(* CODESYS project Alarming.library
   Company: Ziga Javornik
   DefaultNamespace: ZigaLibs.Alarming
   Version: 0.0.3.1
   Placeholder: ZigaLibs.Alarming
   Author: Ziga Javornik
   Description: A library for alarm management. Uses ZigaLibs_Logging to create the alarm logs files.
   Title: ZigaLibs.Alarming

Project tree, tasks and I/O mapping:
  libraries: Tc2_Standard, 3.4.5.0 (Beckhoff Automation GmbH); Tc2_System, 3.6.4.0 (Beckhoff Automation GmbH); Tc2_Utilities, * (Beckhoff Automation GmbH); Tc3_Module, 3.4.5.0 (Beckhoff Automation GmbH); TcUnit, 1.3.1 (www.tcunit.org); ZigaLibs.Core, 0.0.3.7 (Ziga Javornik); ZigaLibs.Logging, 0.0.4.1 (Ziga Javornik)
  GVLs/
  SOURCE/
    AlarmManager/
      Actions - fluent/
        function block FB_AlarmActionBuilder [ST]: Acknowledge, ById, ByName, Deactivate, DoAction, FB_init, Raise, SelectedAlarm
        interface I_AlarmActionBy: ById, ByName
        interface I_AlarmActions: Acknowledge, Deactivate, Raise
      DUTs/
        function block AlarmsArray [ST]: FB_exit, AddNew, Clear, Create, GetPtr, Remove, Set, NumberOfAlarms
        data type ST_AlarmInfo
        data type ST_AlarmTimeInfos
      data type E_AlarmLevel
      function block FB_AlarmManager [ST]: FB_init, AcknowledgeAlarmById, DeactivateAlarmById, RaiseAlarmById, AcknowledgeAlarmByName, DeactivateAlarmByName, RaiseAlarmByName, AcknowledgeAlarm, DeactivateAlarm, DeactivateAllAlarms, GetAlarmIndex, RaiseAlarm, AcknowledgeAllAlarms, Actions, DeleteAlarm, DeleteAll, GetAlarmById, GetAlarmByName, RegisterAlarm, ActiveAlarmsCount, Enable, RegisteredAlarmsCount, UnacknowledgedAlarmsCount
      interface I_AlarmManager: AcknowledgeAllAlarms, Actions, ActiveAlarmsCount, DeleteAlarm, DeleteAll, Enable, GetAlarmById, GetAlarmByName, RegisterAlarm, RegisteredAlarmsCount, UnacknowledgedAlarmsCount
  TESTS/
    Test suites/
      function block FB_AlarmManager_Tests [ST]: Test00_RegisterAlarms, Test01_ActivateNewAlarm_ExpectUnacknowledgedActiveAlarm, Test02_AcknowledgeActiveAlarm_ExpectActiveAcknowledged, Test03_ActivateExistingAlarm_ExpectSameActiveAlarmCount, Test04_DeactivateAlarm_ExpectNotActiveAcknowledged, Test05_AcknowlidgeInactiveAlarm_ExpectAcknowledgedNotActive, Test06_DisableManager_ExpectNoActiveAlarms, Test07_AcknowledgeAllAlarms_ExpectActiveAlarmsUnchanged, Test08_ActivateByName, Test09_DeactivateByName, Test10_AcknowledgeByName, Test11_GetAlarmByName, Test12_GetAlarmById, Test13_ActivateById, Test14_DeactivateById, Test15_AcknowledgeById, Test16_TimeInfos, Test17_RaiseUnexisitngAlarm_ExpectNoNewAlarmsActive, Test18_DeleteAlarm_ExpectPreviousAlarmsStillExist, Test19_DeleteUnexistingAlarm_ExpectNoChangesToExistingAlarms, Test20_DeleteAll
    program PRG_TESTS [ST]
*)

// SOURCE/AlarmManager/DUTs/ST_AlarmInfo
// Alarm information structure, containing all the informations requoired
TYPE ST_AlarmInfo :
STRUCT
	Name			: Tc2_System.T_MaxString;	// Name of the alarm
	Id				: T_ArrayIndexer;			// Id of the alarm
	Message			: Tc2_System.T_MaxString;	// Message of the alarm
	IsActive		: BOOL;						// Active state (TRUE = currently active, FALSE = not active)
	IsAcknowledged	: BOOL;						// Acknowledge state of the alarm
	Level			: E_AlarmLevel;				// Alarm level
	TimeInfos		: ST_AlarmTimeInfos;		// Time informations (activated, acknowldiged, deactivated)
END_STRUCT
END_TYPE

// SOURCE/AlarmManager/DUTs/ST_AlarmTimeInfos
// Provides time information for an alarm
TYPE ST_AlarmTimeInfos :
STRUCT
	Activated		: Tc2_Utilities.TIMESTRUCT;	// Time of alarm activation
	Deactivated		: Tc2_Utilities.TIMESTRUCT;	// Time of alarm deactiovation
	Acknowledged	: Tc2_Utilities.TIMESTRUCT;	// Time of alarm acknowlidgemenet
END_STRUCT
END_TYPE

// SOURCE/AlarmManager/E_AlarmLevel
{attribute 'qualified_only'}
{attribute 'strict'}
// Alarm level enumeration
TYPE E_AlarmLevel :
(
	NONE,
	INFO,
	WARNING,
	ERROR
);
END_TYPE

// SOURCE/AlarmManager/Actions - fluent/FB_AlarmActionBuilder
FUNCTION_BLOCK INTERNAL FB_AlarmActionBuilder IMPLEMENTS I_AlarmActionBy, I_AlarmActions
VAR
	_alarmAction 	: (ACTION_ACKNOWLEDGE, ACTTION_RAISE, ACTION_DEACTIVATE);
	_selectedAlarm	: REFERENCE TO ST_AlarmInfo;
	_alarmManager	: REFERENCE TO FB_AlarmManager;
END_VAR

METHOD Acknowledge : I_AlarmActionBy
VAR_INPUT
END_VAR
_alarmAction := ACTION_ACKNOWLEDGE;
Acknowledge := THIS^;
END_METHOD

// Executes the action by looking for the alarm with the provided ID
METHOD ById
VAR_INPUT
	Id	: T_ArrayIndexer;
END_VAR
VAR
	i	: T_ArrayIndexer;
END_VAR
IF NOT __ISVALIDREF(_alarmManager.GetAlarmById(Id)) THEN
	RETURN;
END_IF

_selectedAlarm REF= _alarmManager.GetAlarmById(Id);
DoAction();
END_METHOD

// Executes the action by looking for the alarm with the provided name
METHOD ByName
VAR_INPUT
	name	: Tc2_System.T_MaxString;
END_VAR

VAR_INST
	i	: T_ArrayIndexer;
END_VAR
IF NOT __ISVALIDREF(_alarmManager.GetAlarmByName(name)) THEN
	RETURN;
END_IF
_selectedAlarm REF= _alarmManager.GetAlarmByName(name);
DoAction();
END_METHOD

METHOD Deactivate : I_AlarmActionBy
VAR_INPUT
END_VAR
_alarmAction := ACTION_DEACTIVATE;
Deactivate := THIS^;
END_METHOD

METHOD PRIVATE DoAction
CASE _alarmAction OF
	ACTION_ACKNOWLEDGE:
		_alarmManager.AcknowledgeAlarm(_selectedAlarm);
	ACTTION_RAISE:
		_alarmManager.RaiseAlarm(_selectedAlarm);
	ACTION_DEACTIVATE:
		_alarmManager.DeactivateAlarm(_selectedAlarm);
END_CASE
END_METHOD

METHOD FB_init : BOOL
VAR_INPUT
	bInitRetains : BOOL; // if TRUE, the retain variables are initialized (warm start / cold start)
	bInCopyCode : BOOL;  // if TRUE, the instance afterwards gets moved into the copy code (online change)
	alarmManager	: REFERENCE TO FB_AlarmManager;
END_VAR
_alarmManager REF= alarmManager;
END_METHOD

METHOD Raise : I_AlarmActionBy
VAR_INPUT
END_VAR
_alarmAction := ACTTION_RAISE;
Raise := THIS^;
END_METHOD

PROPERTY SelectedAlarm : REFERENCE TO ST_AlarmInfo
GET
END_GET
END_PROPERTY

END_FUNCTION_BLOCK

// SOURCE/AlarmManager/Actions - fluent/I_AlarmActionBy
INTERFACE I_AlarmActionBy

// Executes the action by looking for the alarm with the provided ID
METHOD ById
VAR_INPUT
	Id	: T_ArrayIndexer;
END_VAR
END_METHOD

// Executes the action by looking for the alarm with the provided name
METHOD ByName
VAR_INPUT
	name	: Tc2_System.T_MaxString;
END_VAR
END_METHOD

END_INTERFACE

// SOURCE/AlarmManager/Actions - fluent/I_AlarmActions
INTERFACE I_AlarmActions

METHOD Acknowledge : I_AlarmActionBy
VAR_INPUT
END_VAR
END_METHOD

METHOD Deactivate : I_AlarmActionBy
VAR_INPUT
END_VAR
END_METHOD

METHOD Raise : I_AlarmActionBy
VAR_INPUT
END_VAR
END_METHOD

END_INTERFACE

// SOURCE/AlarmManager/FB_AlarmManager
(* 
Alarm manager function block. 
The body does not contain any logic, this it does not require being called.

====================================================
Constructor template:

(enable : , // Enables alarm generation
logger : , // If you do not want logging, simply set this variable to 0, internal checks will ommit any logging.
timeProvider : ); // Date time provider.*)

{attribute 'no_explicit_call' := 'Body contains no logic, calling methods only allowed.'}
FUNCTION_BLOCK FB_AlarmManager IMPLEMENTS I_AlarmManager

VAR
	_enable						: BOOL;
	_stringBuilder				: ZigaLibs_Core.FB_StringBuilder;
	_dateTime					: ZigaLibs_Core.I_LocalSystemTimeProvider;
	_activeAlarmCount			: UINT;
	_logger						: REFERENCE TO ZigaLibs_Logging.I_Logger; // If provided, logging will be used.
	_emptyAlarm					: ST_AlarmInfo;
	_registeredAlarmsCount		: UDINT;
	_alarmActionBuilder			: FB_AlarmActionBuilder(THIS^);
	_alarms						: AlarmsArray;
END_VAR

METHOD FB_init : BOOL
VAR_INPUT
	bInitRetains 	: BOOL; // if TRUE, the retain variables are initialized (warm start / cold start)
	bInCopyCode 	: BOOL;  // if TRUE, the instance afterwards gets moved into the copy code (online change)
	enable			: BOOL;	// Enables alarm generation
	logger			: REFERENCE TO ZigaLibs_Logging.I_Logger; // If you do not want logging, simply set this variable to 0, internal checks will ommit any logging.
	timeProvider	: ZigaLibs_Core.I_LocalSystemTimeProvider;	// Date time provider.
END_VAR
_enable := enable;
_logger REF= logger;
_dateTime := timeProvider;
END_METHOD

(* Acknowledges the alarm with the provided id*)
METHOD INTERNAL AcknowledgeAlarmById
VAR_INPUT
	nId	: T_ArrayIndexer;
END_VAR

VAR
	foundAlarm	: ST_AlarmInfo;
END_VAR
IF NOT __ISVALIDREF(GetAlarmById(nID := nId)) THEN
	RETURN;
END_IF

foundAlarm := GetAlarmById(nID := nId);
IF foundAlarm.Id = nId THEN
	AcknowledgeAlarm(alarm := GetAlarmById(nID := nId));
	RETURN;
END_IF
END_METHOD

(* Deactivates the alarm with the provided Id (if it exists).*)
METHOD INTERNAL DeactivateAlarmById
VAR_INPUT
	(* Alarm id to be deactivated.*)
	nId	: T_ArrayIndexer;
END_VAR

VAR
	foundAlarm	 : ST_AlarmInfo;
END_VAR
IF NOT __ISVALIDREF(GetAlarmById(nID := nId)) THEN
	RETURN;
END_IF

foundAlarm := GetAlarmById(nID := nId);

IF foundAlarm.Id = nId THEN
	DeactivateAlarm(alarm := GetAlarmById(nID := nId));
	RETURN;
END_IF
END_METHOD

(* Activates the alarm with the provided Id (if it exists)*)
METHOD INTERNAL RaiseAlarmById
VAR_INPUT
	(* Alarm id to be activated*)
	nId	: T_ArrayIndexer;
END_VAR

VAR
	foundAlarm	 : ST_AlarmInfo;
END_VAR
IF NOT __ISVALIDREF(GetAlarmById(nID := nId)) THEN
	RETURN;
END_IF

foundAlarm := GetAlarmById(nID := nId);
IF foundAlarm.Id = nId THEN
	RaiseAlarm(alarm := GetAlarmById(nID := nId));
	RETURN;
END_IF
END_METHOD

(* Acknowledges the alarm with the provided name.*)
METHOD INTERNAL AcknowledgeAlarmByName
VAR_INPUT
	sName	: Tc2_System.T_MaxString;
END_VAR

VAR
	foundAlarm	: ST_AlarmInfo;
END_VAR
IF NOT __ISVALIDREF(GetAlarmByName(sName := sName)) THEN
	RETURN;
END_IF

foundAlarm := GetAlarmByName(sName := sName);
IF foundAlarm.Name = sName THEN
	AcknowledgeAlarm(alarm := GetAlarmByName(sName := sName));
	RETURN;
END_IF
END_METHOD

(* Deactivates the alarm with the provided name (if it exists)*)
METHOD INTERNAL DeactivateAlarmByName
VAR_INPUT
	(* Alarm name to be deactivated.*)
	sName	: Tc2_System.T_MaxString;
END_VAR

VAR
	foundAlarm	 : ST_AlarmInfo;
END_VAR
IF NOT __ISVALIDREF(GetAlarmByName(sName := sName)) THEN
	RETURN;
END_IF

foundAlarm := GetAlarmByName(sName := sName);
IF foundAlarm.Name = sName THEN
	DeactivateAlarm(alarm := GetAlarmByName(sName := sName));
	RETURN;
END_IF
END_METHOD

(* Activates the alarm with the provided name*)
METHOD INTERNAL RaiseAlarmByName
VAR_INPUT
	(* Alarm name to be actived*)
	sName	: Tc2_System.T_MaxString;
END_VAR

VAR
	foundAlarm	 : ST_AlarmInfo;
END_VAR
IF NOT __ISVALIDREF(GetAlarmByName(sName := sName)) THEN
	RETURN;
END_IF

foundAlarm := GetAlarmByName(sName := sName);
IF foundAlarm.Name = sName THEN
	RaiseAlarm(alarm := GetAlarmByName(sName := sName));
	RETURN;
END_IF
END_METHOD

METHOD INTERNAL AcknowledgeAlarm
VAR_INPUT
	alarm : REFERENCE TO ST_AlarmInfo;
END_VAR
IF alarm.IsAcknowledged THEN
	RETURN;
END_IF

alarm.IsAcknowledged := TRUE;
alarm.TimeInfos.Acknowledged := _dateTime.CurrentTime.Value;

IF __ISVALIDREF(_logger) THEN 
	_logger.LogInfo(_stringBuilder.Reset()
		.AddString('Alarm ')
		.AddWithDblQuotationMarks(str := alarm.Name)
		.AddString(' with Id ')
		.AddWithDblQuotationMarks(str := TO_STRING(alarm.Id))
		.AddString(' acknowledged.')
		.Create());
END_IF
END_METHOD

METHOD INTERNAL DeactivateAlarm
VAR_INPUT
	alarm : REFERENCE TO ST_AlarmInfo;
END_VAR
IF NOT alarm.IsActive THEN
	RETURN;
END_IF

alarm.IsActive := FALSE;
alarm.TimeInfos.Deactivated := _dateTime.CurrentTime.Value;
_activeAlarmCount := _activeAlarmCount - 1;

IF __ISVALIDREF(_logger) THEN
	_logger.LogInfo(_stringBuilder
		.Reset()
		.AddString('Alarm ')
		.AddWithDblQuotationMarks(str := alarm.Name)
		.AddString(' with Id ')
		.AddWithDblQuotationMarks(str := TO_STRING(alarm.Id))
		.AddString(' deactivated.')
		.Create());
END_IF
END_METHOD

METHOD PRIVATE DeactivateAllAlarms

VAR
	alarmIndex	: T_ArrayIndexer;
END_VAR
FOR alarmIndex := 0 TO _alarms.NumberOfAlarms BY 1 DO
	IF _alarms.GetPtr(alarmIndex) <> 0 AND_THEN _alarms.GetPtr(alarmIndex)^.IsActive THEN
		DeactivateAlarm(_alarms.GetPtr(alarmIndex)^);
	END_IF
END_FOR
END_METHOD

METHOD PRIVATE GetAlarmIndex : DINT
VAR_INPUT
	id	: DINT;
END_VAR
VAR_OUTPUT
	exists	: BOOL;
END_VAR
VAR
	alarmIndex	: DINT;
	alarmPtr	: POINTER TO ST_AlarmInfo;
END_VAR
FOR alarmIndex := 0 TO _alarms.NumberOfAlarms - 1 BY 1 DO
	alarmPtr := _alarms.GetPtr(alarmIndex);
	IF alarmPtr <> 0 AND_THEN alarmPtr^.Id = id THEN 
		GetAlarmIndex := alarmIndex;
		exists := TRUE;
		RETURN;
	END_IF
END_FOR
END_METHOD

METHOD INTERNAL RaiseAlarm
VAR_INPUT
	alarm : REFERENCE TO ST_AlarmInfo;
END_VAR
VAR
	message	: Tc2_System.T_MaxString;
END_VAR
IF alarm.IsActive OR NOT _enable THEN
	RETURN;
END_IF

_activeAlarmCount := _activeAlarmCount + 1;
alarm.IsActive := TRUE;
alarm.IsAcknowledged := FALSE;
Tc2_System.MEMSET(
	destAddr := ADR(alarm.TimeInfos),
	fillByte := 0,
	n := SIZEOF(alarm.TimeInfos));
	
alarm.TimeInfos.Activated := _dateTime.CurrentTime.Value;

IF __ISVALIDREF(_logger) THEN
	message := _stringBuilder.Reset()
		.AddString('Alarm ')
		.AddWithDblQuotationMarks(str := alarm.Name)
		.AddString(' with Id ')
		.AddWithDblQuotationMarks(str := TO_STRING(alarm.Id))
		.AddString(' actived! ')
		.AddString(alarm.Message)
		.Create();
		
	CASE alarm.Level OF 
		E_AlarmLevel.NONE: _logger.LogDefault(message := message);
		E_AlarmLevel.INFO: _logger.LogInfo(message := message);
		E_AlarmLevel.WARNING: _logger.LogWarning(message := message);
		E_AlarmLevel.ERROR: _logger.LogError(message := message);
	END_CASE
END_IF
END_METHOD

(* Acknowledges all uacknowledged alarms.*)
METHOD AcknowledgeAllAlarms
VAR
	alarmIndex	: T_ArrayIndexer;
END_VAR
FOR alarmIndex := 0 TO _alarms.NumberOfAlarms - 1 BY 1 DO
	IF _alarms.GetPtr(alarmIndex) <> 0 THEN 
		AcknowledgeAlarm(_alarms.GetPtr(alarmIndex)^);
	END_IF
END_FOR
END_METHOD

// Provides access to action builder with fluent approach.
METHOD PUBLIC Actions : I_AlarmActions
VAR_INPUT
END_VAR
Actions := _alarmActionBuilder;
END_METHOD

(* Deletes the alarm with the provided id.*)
METHOD DeleteAlarm
VAR_INPUT
	id	: DINT;
END_VAR
VAR
	exists	: BOOL;
	index	: DINT;
	alarm	: POINTER TO ST_AlarmInfo;
END_VAR
index := THIS^.GetAlarmIndex(id, exists => exists);
IF exists THEN
	alarm := _alarms.GetPtr(index);
	IF alarm^.IsActive THEN
		_activeAlarmCount := _activeAlarmCount - 1;
	END_IF
	_alarms.Remove(index);
END_IF
END_METHOD

(* Deletes all existing alarms from the memory*)
METHOD DeleteAll
_alarms.Clear();
_activeAlarmCount := 0;
END_METHOD

(* Gets the alarm with the provided id. 
 If no mathching alarm exists, an invalid reference will be returned - check by using __ISVALIDREF() for any further operations!.*)
METHOD GetAlarmById : REFERENCE TO ST_AlarmInfo
VAR_INPUT
	(* Id of the alarm.*)
	nID	: T_ArrayIndexer;
END_VAR

VAR
	index		: ZigaLibs_Core.T_ArrayIndexer;
	alarmPtr	: POINTER TO ST_AlarmInfo;
END_VAR
FOR index := 0 TO _alarms.NumberOfAlarms - 1 BY 1 DO
	alarmPtr := _alarms.GetPtr(index);
	IF alarmPtr <> 0 AND_THEN alarmPtr^.Id = nId THEN
		GetAlarmById REF= _alarms.GetPtr(index)^;
		RETURN;
	END_IF
END_FOR
END_METHOD

(* Gets the alarm with the provided name. 
 If no mathching alarm exists, an empty alarm is returned.*)
METHOD GetAlarmByName : REFERENCE TO ST_AlarmInfo
VAR_INPUT
	(* Name of the alarm*)
	sName	: Tc2_System.T_MaxString;
END_VAR

VAR
	index	 : T_ArrayIndexer;
END_VAR
FOR index := 0 TO _alarms.NumberOfAlarms - 1 BY 1 DO
	IF _alarms.GetPtr(index) <> 0 AND_THEN _alarms.GetPtr(index)^.Name = sName THEN
		GetAlarmByName REF= _alarms.GetPtr(index)^;
		RETURN;
	END_IF
END_FOR
END_METHOD

(* Registers a new alarm with the provided information. 
 Returns TRUE if new alarm was registered or false if not (alarm buffer is full or the id already exists)*)
METHOD RegisterAlarm : BOOL
VAR_INPUT
	(* Alarm ID*)
	Id	: T_ArrayIndexer;
	(* Alarm name*)
	Name	: Tc2_System.T_MaxString;
	(* Message when the alarm occurrs*)
	Message	: Tc2_System.T_MaxString;
	(* Alarm level *)
	Level	: E_AlarmLevel;				
END_VAR

VAR
	alarmIndex	: T_ArrayIndexer;
	alarm		:  ST_AlarmInfo;
END_VAR
// IF an alar is found, check the id and return.
IF __ISVALIDREF(GetAlarmById(nID := Id)) AND_THEN GetAlarmById(nID := Id).Id = Id 
THEN
	RETURN;
END_IF

// Create the alarm
alarm.Id := Id;
alarm.Name := Name;
alarm.Message := Message;
alarm.IsAcknowledged := TRUE;
alarm.Level := Level;
_alarms.AddNew(alarm);
RegisterAlarm := TRUE;
END_METHOD

{attribute 'monitoring':='call'}
(* Gets the total count of currently active alarms*)
PROPERTY ActiveAlarmsCount : UINT
GET
ActiveAlarmsCount := _activeAlarmCount;
END_GET
END_PROPERTY

{attribute 'monitoring':='call'}
(* Gets or sets if alarm manager is enabled or not. When disabled, all active alarms will become inactive!*)
PROPERTY Enable : BOOL
GET
Enable := _enable;
END_GET
SET
IF NOT Enable AND _enable THEN 
	IF __ISVALIDREF(_logger) THEN
		_logger.LogInfo('Alarms are now disabled.');
	END_IF
	DeactivateAllAlarms();
	AcknowledgeAllAlarms();
ELSIF Enable AND NOT _enable THEN
	IF __ISVALIDREF(_logger) THEN
		_logger.LogInfo('Alarms are now enabled.');
	END_IF
END_IF

_enable := Enable;
END_SET
END_PROPERTY

{attribute 'monitoring':='call'}
(* Gets the total number of alarms registered*)
PROPERTY RegisteredAlarmsCount : UDINT
GET
RegisteredAlarmsCount := DINT_TO_UDINT(_alarms.NumberOfAlarms);
END_GET
END_PROPERTY

{attribute 'monitoring':='call'}
(* Gets the current count of alarms that have not yet been acknowledged*)
PROPERTY UnacknowledgedAlarmsCount : UINT
GET
VAR
	alarmIndex		: T_ArrayIndexer;
	maxAlarmIndex	: T_ArrayIndexer;
	count			: UINT;
END_VAR
FOR alarmIndex := 0 TO _alarms.NumberOfAlarms - 1 BY 1 DO
	IF _alarms.GetPtr(alarmIndex) <> 0 AND_THEN NOT _alarms.GetPtr(alarmIndex)^.IsAcknowledged THEN
		count := count + 1;
	END_IF
END_FOR

UnacknowledgedAlarmsCount := count;
END_GET
END_PROPERTY

END_FUNCTION_BLOCK

// SOURCE/AlarmManager/I_AlarmManager
INTERFACE I_AlarmManager

// Acknowledges all uacknowledged alarms.
METHOD AcknowledgeAllAlarms
END_METHOD

// Provides access to action builder with fluent approach.
METHOD PUBLIC Actions : I_AlarmActions
VAR_INPUT
END_VAR
END_METHOD

{attribute 'monitoring':='call'}
// Gets the total count of currently active alarms
PROPERTY ActiveAlarmsCount : UINT
GET
END_GET
END_PROPERTY

// Deletes the alarm with the provided id.
METHOD DeleteAlarm
VAR_INPUT
	id	: DINT;
END_VAR
END_METHOD

// Deletes all existing alarms from the memory
METHOD DeleteAll
END_METHOD

{attribute 'monitoring':='call'}
// Gets or sets if alarm manager is enabled or not. When disabled, all active alarms will become inactive!
PROPERTY Enable : BOOL
GET
END_GET
SET
END_SET
END_PROPERTY

(* Gets the alarm with the provided id. 
 If no mathching alarm exists, an invalid reference will be returned - check by using __ISVALIDREF() for any further operations!.*)
METHOD GetAlarmById : REFERENCE TO ST_AlarmInfo
VAR_INPUT
	nID		: T_ArrayIndexer;	// Id of the alarm.
END_VAR
END_METHOD

// Gets the alarm with the provided name. 
// IF no mathching alarm exists, an invalid REFERENCE will be returned - check BY using __ISVALIDREF() FOR ANY further operations!.*)
METHOD GetAlarmByName : REFERENCE TO ST_AlarmInfo
VAR_INPUT
	sName	: Tc2_System.T_MaxString;	// Name of the alarm
END_VAR
END_METHOD

// Registers a new alarm with the provided information. 
// Returns TRUE if new alarm was registered or false if not
// Possible reasons for fail:
// - alarm buffer is full
// - the id already exists)
METHOD RegisterAlarm : BOOL
VAR_INPUT
	Id		: T_ArrayIndexer;			// Alarm ID
	Name	: Tc2_System.T_MaxString;	// Alarm name
	Message	: Tc2_System.T_MaxString;	// Message when the alarm occurrs
	Level	: E_AlarmLevel;				// Alarm level
END_VAR
END_METHOD

{attribute 'monitoring':='call'}
// Gets the total number of alarms registered
PROPERTY RegisteredAlarmsCount : UDINT
GET
END_GET
END_PROPERTY

{attribute 'monitoring':='call'}
// Gets the current count of alarms that have not yet been acknowledged
PROPERTY UnacknowledgedAlarmsCount : UINT
GET
END_GET
END_PROPERTY

END_INTERFACE

// SOURCE/AlarmManager/DUTs/AlarmsArray
// A dynamic collection of alarms as ST_AlarmInfo
FUNCTION_BLOCK AlarmsArray
VAR_INPUT
END_VAR
VAR_OUTPUT
END_VAR
VAR
	_malloc	: ZigaLibs_Core.FB_Malloc(0,0);
END_VAR

METHOD FB_exit : BOOL
VAR_INPUT
	bInCopyCode : BOOL; // if TRUE, the exit method is called for exiting an instance that is copied afterwards (online change).
END_VAR
_malloc.Free();
END_METHOD

// Adds a new alarm defintition to the collection
METHOD AddNew
VAR_INPUT
	alarm	: ST_AlarmInfo;
END_VAR
IF NOT _malloc.IsAllocated THEN
	THIS^.Create(1);
	THIS^.GetPtr(0)^ := alarm;
ELSE
	_malloc.Expand(1);
	_malloc.Set(_malloc.Properties.NumberOfElements - 1, alarm);
END_IF
END_METHOD

// Clear the entire collection of alarms
METHOD Clear
VAR_INPUT
END_VAR
_malloc.Free();
END_METHOD

// Creates a number of alarms defined by the count value
METHOD Create : BOOL
VAR_INPUT
	count	: dint;
END_VAR
Create := _malloc.Allocate(SIZEOF(ST_AlarmInfo), count);
END_METHOD

// Gets the pointer to the desired ST_AlarmInfo info at index
METHOD GetPtr : POINTER TO ST_AlarmInfo
VAR_INPUT
	index	: DINT;
END_VAR
GetPtr := _malloc.GetPtr(index);
END_METHOD

// Romves an alarm at the provided index
METHOD Remove
VAR_INPUT
	index	: DINT;
END_VAR
_malloc.Remove(index);
END_METHOD

// Sets the alarm at the index to the value provided in the alarm
METHOD Set : BOOL
VAR_INPUT
	index	: DINT;
	alarm	: REFERENCE TO ST_AlarmInfo;
END_VAR
Set := _malloc.Set(index := index, value := alarm);
END_METHOD

{attribute 'monitoring':='call'}
// Gets the total number of alarms in the collection
PROPERTY NumberOfAlarms : DINT
GET
NumberOfAlarms := _malloc.Properties.NumberOfElements;
END_GET
END_PROPERTY

END_FUNCTION_BLOCK

// TESTS/Test suites/FB_AlarmManager_Tests
FUNCTION_BLOCK INTERNAL FB_AlarmManager_Tests EXTENDS FB_TestSuite
VAR
	_dateTime	: ZigaLibs_Core.FB_LocalSystemTimeProvider;
	_alarmManager : FB_AlarmManager(
		enable := TRUE, // [BOOL] - Enables alarm generation
		logger := 0, // [REFERENCE TO ZigaLibs_Core.I_LoggerEx] - optional, logger.
		timeProvider := _dateTime); //[ZigaLibs_Core.I_LocalSystemTimeProvider] - required, date time provider.
END_VAR

_dateTime();
Test00_RegisterAlarms();
Test01_ActivateNewAlarm_ExpectUnacknowledgedActiveAlarm();
Test02_AcknowledgeActiveAlarm_ExpectActiveAcknowledged();
Test03_ActivateExistingAlarm_ExpectSameActiveAlarmCount();
Test04_DeactivateAlarm_ExpectNotActiveAcknowledged();
Test05_AcknowlidgeInactiveAlarm_ExpectAcknowledgedNotActive();
Test06_DisableManager_ExpectNoActiveAlarms();
Test07_AcknowledgeAllAlarms_ExpectActiveAlarmsUnchanged();
Test08_ActivateByName();
Test09_DeactivateByName();
Test10_AcknowledgeByName();
Test11_GetAlarmByName();
Test12_GetAlarmById();
Test13_ActivateById();
Test14_DeactivateById();
Test15_AcknowledgeById();
Test16_TimeInfos();
Test17_RaiseUnexisitngAlarm_ExpectNoNewAlarmsActive();
Test18_DeleteAlarm_ExpectPreviousAlarmsStillExist();
Test19_DeleteUnexistingAlarm_ExpectNoChangesToExistingAlarms();
Test20_DeleteAll();

METHOD Test00_RegisterAlarms
VAR_INPUT
END_VAR

VAR
	addAlarmIndex	: T_ArrayIndexer;
	alarm			: ST_AlarmInfo;
END_VAR
IF TcUnit.TEST_ORDERED('Test00_RegisterAlarms') THEN
	AssertEquals_UDINT(
		Actual := _alarmManager.RegisteredAlarmsCount,
		Expected := 0,
		Message := 'Before registering any alarms, the Registered count should be 0.');
	
	FOR addAlarmIndex := 1 TO 100 BY 1 DO
		AssertTrue(
			Condition := _alarmManager.RegisterAlarm(
				Id := addAlarmIndex,
				Message := Tc2_Standard.CONCAT('Alarm message', TO_STRING(addAlarmIndex)),
				Name := Tc2_Standard.CONCAT('Alarm name', TO_STRING(addAlarmIndex)),
				Level := E_AlarmLevel.INFO),
			Message := 'Registering alarm failed.');
			
		AssertEquals_UDINT(
			Actual := _alarmManager.RegisteredAlarmsCount,
			Expected := DINT_TO_UDINT(addAlarmIndex),
			Message := 'Registered alarm count is incorrect.');
			
		alarm := _alarmManager.GetAlarmById(nID := addAlarmIndex);
		AssertTrue(
			Condition := alarm.IsAcknowledged,
			Message := 'Newly registered alarm should be acknowledged by default, when created.');
	END_FOR
	
	AssertFalse(
		Condition := _alarmManager.RegisterAlarm(
			Id := 22,
			Message := CONCAT('Alarm message', TO_STRING(addAlarmIndex - 1)),
			Name := CONCAT('Alarm name', TO_STRING(addAlarmIndex - 1)),
			Level := E_AlarmLevel.INFO),
		Message := 'Registering an alarm with an existing id should not be possible.');
	
		
	TcUnit.TEST_FINISHED();
END_IF
END_METHOD

METHOD Test01_ActivateNewAlarm_ExpectUnacknowledgedActiveAlarm
VAR_INPUT
END_VAR

VAR
	currentAlarm	: ST_AlarmInfo;
END_VAR
IF TcUnit.TEST_ORDERED('Test01_ActivateNewAlarm_ExpectUnacknowledgedActiveAlarm') THEN
	_alarmManager.RaiseAlarmById(10);
	currentAlarm := _alarmManager.GetAlarmById(10);
	
	AssertEquals_BOOL(
		Actual := currentAlarm.IsActive,
		Expected := TRUE,
		Message := 'Alarm activation failed.');
		
	AssertEquals_BOOL(
		Actual := currentAlarm.IsAcknowledged,
		Expected := FALSE,
		Message := 'Newly activated alarm should not be acknowledged.');	
	
		
	AssertEquals_UINT(
		Actual := _alarmManager.ActiveAlarmsCount,
		Expected := 1,
		Message := 'Active alarm count is incorrect.');
	
	AssertEquals_UINT(
		Actual := _alarmManager.UnacknowledgedAlarmsCount,
		Expected := 1,
		Message := 'Unacknowledged alarm count is incorrect.');
		
	TcUnit.TEST_FINISHED();
END_IF
END_METHOD

METHOD Test02_AcknowledgeActiveAlarm_ExpectActiveAcknowledged
VAR_INPUT
END_VAR
IF TcUnit.TEST_ORDERED('Test02_AcknowledgeActiveAlarm_ExpectActiveAcknowledged') THEN

	_alarmManager.AcknowledgeAlarmById(10);
	
	AssertEquals_BOOL(
		Actual := _alarmManager.GetAlarmById(10).IsActive,
		Expected := TRUE,
		Message := 'Alarm activation failed.');
		
	AssertEquals_BOOL(
		Actual := _alarmManager.GetAlarmById(10).IsAcknowledged,
		Expected := TRUE,
		Message := 'Acknowlidging active alarm failed.');	
	
	TcUnit.TEST_FINISHED();
END_IF
END_METHOD

METHOD Test03_ActivateExistingAlarm_ExpectSameActiveAlarmCount
VAR_INPUT
END_VAR
IF TcUnit.TEST_ORDERED('Test03_ActivateExistingAlarm_ExpectSameActiveAlarmCount') THEN
	_alarmManager.RaiseAlarmById(10);	
	AssertEquals_BOOL(
		Actual := _alarmManager.GetAlarmById(10).IsActive,
		Expected := TRUE,
		Message := 'Alarm activation failed.');
		
	AssertEquals_BOOL(
		Actual := _alarmManager.GetAlarmById(10).IsAcknowledged,
		Expected := TRUE,
		Message := 'Already acknowledged alarm should not be acknowledged when activating the alarm while it is already active.');	
	
		
	AssertEquals_UINT(
		Actual := _alarmManager.ActiveAlarmsCount,
		Expected := 1,
		Message := 'Active alarm count is incorrect.');
	
	AssertEquals_UINT(
		Actual := _alarmManager.UnacknowledgedAlarmsCount,
		Expected := 0,
		Message := 'Activating acknowledged and already active alarm should not cause the alarm to be unacknowledged..');
		
	TcUnit.TEST_FINISHED();
END_IF
END_METHOD

METHOD Test04_DeactivateAlarm_ExpectNotActiveAcknowledged
VAR_INPUT
END_VAR
IF TcUnit.TEST_ORDERED('Test04_DeactivateAlarm_ExpectNotActiveAcknowledged') THEN
	_alarmManager.DeactivateAlarmById(10);
	
	AssertFalse(
		Condition := _alarmManager.GetAlarmById(10).IsActive,
		Message := 'Alarm deactivation failed.');
		
	AssertTrue(
		Condition := _alarmManager.GetAlarmById(10).IsAcknowledged,
		Message := 'Alarm deactivation should not acknowledge the alarm.');	
		
	AssertEquals_UINT(
		Actual := _alarmManager.ActiveAlarmsCount,
		Expected := 0,
		Message := 'Active alarm count is incorrect.');
	
	AssertEquals_UINT(
		Actual := _alarmManager.UnacknowledgedAlarmsCount,
		Expected := 0,
		Message := 'Unacknowledged alarm count is incorrect.');
		
	TcUnit.TEST_FINISHED();
END_IF
END_METHOD

METHOD Test05_AcknowlidgeInactiveAlarm_ExpectAcknowledgedNotActive
VAR_INPUT
END_VAR
IF TcUnit.TEST_ORDERED('Test05_AcknowlidgeInactiveAlarm_ExpectAcknowledgedNotActive') THEN
	_alarmManager.AcknowledgeAlarmById(10);
	
	AssertEquals_BOOL(
		Actual := _alarmManager.GetAlarmById(10).IsActive,
		Expected := FALSE,
		Message := 'Alarm deactivation failed.');
		
	AssertEquals_BOOL(
		Actual := _alarmManager.GetAlarmById(10).IsAcknowledged,
		Expected := TRUE,
		Message := 'Acknowlidging alarm failed.');	
	
		
	AssertEquals_UINT(
		Actual := _alarmManager.ActiveAlarmsCount,
		Expected := 0,
		Message := 'Active alarm count is incorrect.');
	
	AssertEquals_UINT(
		Actual := _alarmManager.UnacknowledgedAlarmsCount,
		Expected := 0,
		Message := 'Unacknowledged alarm count is incorrect.');
		
	TcUnit.TEST_FINISHED();
END_IF
END_METHOD

METHOD Test06_DisableManager_ExpectNoActiveAlarms
VAR_INPUT
END_VAR
VAR
	n	: T_ArrayIndexer;
END_VAR
IF TcUnit.TEST_ORDERED('Test06_DisableManager_ExpectNoActiveAlarms') THEN
	FOR n := 1 TO 40 BY 1 DO
		_alarmManager.RaiseAlarmById(n);
	END_FOR
	
	AssertEquals_UINT(
		Expected := 40,
		Actual := _alarmManager.ActiveAlarmsCount,
		Message := 'There should only be 40 active alarms at this point.');
			
	_alarmManager.Enable := FALSE;
	
	AssertEquals_UINT(
		Expected := 0,
		Actual := _alarmManager.ActiveAlarmsCount,
		Message := 'Disabling the manager should result in all of the alarms being inactive.');
	
	_alarmManager.Enable := TRUE;
	
	TcUnit.TEST_FINISHED();
END_IF
END_METHOD

METHOD Test07_AcknowledgeAllAlarms_ExpectActiveAlarmsUnchanged
VAR_INPUT
END_VAR

VAR
	n : T_ArrayIndexer;
	fbAlarmManager	: FB_AlarmManager(
		enable := TRUE, // [BOOL] - Enables alarm generation
		logger := 0, // [REFERENCE TO ZigaLibs_Core.I_LoggerEx] - optional, logger.
		timeProvider := _dateTime); //[ZigaLibs_Core.I_LocalSystemTimeProvider] - required, date time provider.
	arrAlarms		: ARRAY[0..60] OF ST_AlarmInfo;
END_VAR
IF TcUnit.TEST_ORDERED('Test07_AcknowledgeAllAlarms_ExpectActiveAlarmsUnchanged') THEN
	FOR n := 1 TO 40 BY 1 DO
		fbAlarmManager.RegisterAlarm(n, TO_STRING(n), '', E_AlarmLevel.INFO);
		fbAlarmManager.RaiseAlarmById(n);
	END_FOR
	
	AssertEquals_UINT(
		Expected := 40,
		Actual := fbAlarmManager.ActiveAlarmsCount,
		Message := 'There should only be 40 active alarms at this point.');
			
	fbAlarmManager.AcknowledgeAllAlarms();
	
	AssertEquals_UINT(
		Expected := 0,
		Actual := fbAlarmManager.UnacknowledgedAlarmsCount,
		Message := 'Acknowlidging all alarms should result in no unacknowledged alarms.');
	
	AssertEquals_UINT(
		Expected := 40,
		Actual := fbAlarmManager.ActiveAlarmsCount,
		Message := 'There should still be 40 active alarms, acknowlidning alarms should not affect alarm state.');
		
	TcUnit.TEST_FINISHED();
END_IF
END_METHOD

METHOD Test08_ActivateByName
VAR_INPUT
END_VAR
IF TcUnit.TEST_ORDERED('Test08_ActivateByName') THEN
	// Reset all alarms this way
	_alarmManager.Enable := FALSE;
	_alarmManager.Enable := TRUE;
	
	_alarmManager.RaiseAlarmByName('Alarm name10');
	
	AssertTrue(
		Condition := _alarmManager.GetAlarmByName('Alarm name10').IsActive,
		Message := 'Activating alarm by name failed.');
	
	AssertFalse(
		Condition := _alarmManager.GetAlarmByName('Alarm name10').IsAcknowledged,
		Message := 'Alarm shold be unacknowledged.');
		
	_alarmManager.DeactivateAlarmByName('Alarm name10');
	_alarmManager.AcknowledgeAlarmByName('Alarm name10');
	
	_alarmManager.Actions()
		.Raise()
		.ByName('Alarm name10');
	
	AssertTrue(
		Condition := _alarmManager.GetAlarmByName('Alarm name10').IsActive,
		Message := 'Fluent - Activating alarm by name failed.');
	
	AssertFalse(
		Condition := _alarmManager.GetAlarmByName('Alarm name10').IsAcknowledged,
		Message := 'Fluent - Alarm shold be unacknowledged.');
		
	TcUnit.TEST_FINISHED();
END_IF
END_METHOD

METHOD Test09_DeactivateByName
VAR_INPUT
END_VAR
IF TcUnit.TEST_ORDERED('Test09_DeactivateByName') THEN
	_alarmManager.DeactivateAlarmByName('Alarm name10');
	AssertFalse(
		Condition := _alarmManager.GetAlarmByName('Alarm name10').IsActive,
		Message := 'Deactivate alarm by name failed.');
	
	AssertFalse(
		Condition := _alarmManager.GetAlarmByName('Alarm name10').IsAcknowledged,
		Message := 'Alarm shold be unacknowledged.');
		
	_alarmManager.RaiseAlarmByName('Alarm name10');
		
	_alarmManager.Actions()
		.Deactivate()
		.ByName('Alarm name10');
	
	AssertFalse(
		Condition := _alarmManager.GetAlarmByName('Alarm name10').IsActive,
		Message := 'Fluent - deactivating alarm by name failed.');
	
	AssertFalse(
		Condition := _alarmManager.GetAlarmByName('Alarm name10').IsAcknowledged,
		Message := 'Fluent - Alarm shold be unacknowledged.');
		
	TcUnit.TEST_FINISHED();
END_IF
END_METHOD

METHOD Test10_AcknowledgeByName
VAR_INPUT
END_VAR
IF TcUnit.TEST_ORDERED('Test10_AcknowledgeByName') THEN
	_alarmManager.AcknowledgeAlarmByName('Alarm name10');
	
	AssertTrue(
		Condition := _alarmManager.GetAlarmByName('Alarm name10').IsAcknowledged,
		Message := 'Alarm shold be acknowledged.');
	
		
	_alarmManager.Actions().Raise().ByName('Alarm name10');
	_alarmManager.Actions().Deactivate().ByName('Alarm name10');
	_alarmManager.Actions().Acknowledge().ByName('Alarm name10');
	AssertTrue(
		Condition := _alarmManager.GetAlarmByName('Alarm name10').IsAcknowledged,
		Message := 'Fluent - Alarm shold be acknowledged.');
		
	TcUnit.TEST_FINISHED();
END_IF
END_METHOD

METHOD Test11_GetAlarmByName
VAR_INPUT
END_VAR

VAR_INST
	fbAlarmManager	: FB_AlarmManager(
		enable := TRUE, // [BOOL] - Enables alarm generation
		logger := 0, // [REFERENCE TO ZigaLibs_Core.I_LoggerEx] - optional, logger.
		timeProvider := _dateTime); //[ZigaLibs_Core.I_LocalSystemTimeProvider] - required, date time provider.
	i				: T_ArrayIndexer;
END_VAR
IF TcUnit.TEST_ORDERED('Test11_GetAlarmByName') THEN
	FOR i := 1 TO 11 BY 1 DO
		fbAlarmManager.RegisterAlarm(i, TO_STRING(i), '',E_AlarmLevel.INFO);
		AssertEquals_STRING(
			Actual := fbAlarmManager.GetAlarmByName(sName := TO_STRING(i)).Name,
			Expected := TO_STRING(i),
			Message := CONCAT('Getting alarm by name failed for alarm', TO_STRING(i)));	
	END_FOR
	
	AssertFalse(
		Condition := __ISVALIDREF(fbAlarmManager.GetAlarmByName('Surely I dont exist...')),
		Message := 'Fetching an alarm by non existing name should return invalid reference.');
	
	TcUnit.TEST_FINISHED();
END_IF
END_METHOD

METHOD Test12_GetAlarmById
VAR_INPUT
END_VAR
VAR_INST
	fbAlarmManager	: FB_AlarmManager(
		enable := TRUE, // [BOOL] - Enables alarm generation
		logger := 0, // [REFERENCE TO ZigaLibs_Core.I_LoggerEx] - optional, logger.
		timeProvider := _dateTime); //[ZigaLibs_Core.I_LocalSystemTimeProvider] - required, date time provider.
	i	: T_ArrayIndexer;
END_VAR
IF TcUnit.TEST_ORDERED('Test12_GetAlarmById') THEN
	FOR i := 1 TO 11 BY 1 DO
		fbAlarmManager.RegisterAlarm(i, TO_STRING(i), '', E_AlarmLevel.INFO);
		AssertEquals_DINT(
			Actual := fbAlarmManager.GetAlarmById(i).Id,
			Expected := i,
			Message := CONCAT('Getting alarm by id failed for alarm', TO_STRING(i)));	
	END_FOR
	
	TcUnit.TEST_FINISHED();
END_IF
END_METHOD

METHOD Test13_ActivateById
VAR_INPUT
END_VAR
IF TcUnit.TEST_ORDERED('Test13_ActivateById') THEN
	// Reset all alarms this way
	_alarmManager.Enable := FALSE;
	_alarmManager.Enable := TRUE;
	
	_alarmManager.RaiseAlarmById(10);
	
	AssertTrue(
		Condition := _alarmManager.GetAlarmById(10).IsActive,
		Message := 'Activating alarm by id failed.');
	
	AssertFalse(
		Condition := _alarmManager.GetAlarmById(10).IsAcknowledged,
		Message := 'Alarm shold be unacknowledged.');
		
	_alarmManager.DeactivateAlarmById(10);
	_alarmManager.AcknowledgeAlarmById(10);
	
	_alarmManager.Actions()
		.Raise()
		.ById(10);
	
	AssertTrue(
		Condition := _alarmManager.GetAlarmById(10).IsActive,
		Message := 'Fluent - Activating alarm by name failed.');
	
	AssertFalse(
		Condition := _alarmManager.GetAlarmById(10).IsAcknowledged,
		Message := 'Fluent - Alarm shold be unacknowledged.');
		
	TcUnit.TEST_FINISHED();
END_IF
END_METHOD

METHOD Test14_DeactivateById
VAR_INPUT
END_VAR
IF TcUnit.TEST_ORDERED('Test14_DeactivateById') THEN
	_alarmManager.DeactivateAlarmById(10);
	AssertFalse(
		Condition := _alarmManager.GetAlarmById(10).IsActive,
		Message := 'Deactivate alarm by name failed.');
	
	AssertFalse(
		Condition := _alarmManager.GetAlarmById(10).IsAcknowledged,
		Message := 'Alarm shold be unacknowledged.');
		
	_alarmManager.RaiseAlarmById(13);
		
	_alarmManager.Actions()
		.Deactivate()
		.ById(13);
	
	AssertFalse(
		Condition := _alarmManager.GetAlarmById(10).IsActive,
		Message := 'Fluent - deactivating alarm by name failed.');
	
	AssertFalse(
		Condition := _alarmManager.GetAlarmById(10).IsAcknowledged,
		Message := 'Fluent - Alarm shold be unacknowledged.');
		
	TcUnit.TEST_FINISHED();
END_IF
END_METHOD

METHOD Test15_AcknowledgeById
VAR_INPUT
END_VAR
IF TcUnit.TEST_ORDERED('Test15_AcknowledgeById') THEN
	_alarmManager.AcknowledgeAlarmById(10);
	
	AssertTrue(
		Condition := _alarmManager.GetAlarmById(10).IsAcknowledged,
		Message := 'Alarm shold be acknowledged.');
	
		
	_alarmManager.Actions().Raise().ById(10);
	_alarmManager.Actions().Deactivate().ById(10);
	_alarmManager.Actions().Acknowledge().ById(10);
	AssertTrue(
		Condition := _alarmManager.GetAlarmById(10).IsAcknowledged,
		Message := 'Fluent - Alarm shold be acknowledged.');
		
	TcUnit.TEST_FINISHED();
END_IF
END_METHOD

METHOD Test16_TimeInfos
VAR_INPUT
END_VAR

VAR_INST
	fbAlarmManager			: FB_AlarmManager(
		enable := TRUE, // [BOOL] - Enables alarm generation
		logger := 0, // [REFERENCE TO ZigaLibs_Core.I_LoggerEx] - optional, logger.
		timeProvider := _dateTime); //[ZigaLibs_Core.I_LocalSystemTimeProvider] - required, date time provider.
	i						: T_ArrayIndexer;
	stTimeStruct			: Tc2_Utilities.TIMESTRUCT;
	stTimeStructActivation	: Tc2_Utilities.TIMESTRUCT;	
	stTimeStructAcnowledge	: Tc2_Utilities.TIMESTRUCT;
	stTimeInfos	: ST_AlarmTimeInfos;
	alarm			: ST_AlarmInfo;
END_VAR
IF TcUnit.TEST_ORDERED('Test16_TimeInfos') THEN
	IF fbAlarmManager._dateTime.CurrentTime.IsValid THEN
		FOR i := 0 TO 10 BY 1 DO
			fbAlarmManager.RegisterAlarm(i,'','', E_AlarmLevel.INFO);
			
			IF NOT __ISVALIDREF(fbAlarmManager.GetAlarmById(i)) THEN
				AssertTrue(Condition := FALSE, 'Creating alarm failed, returned reference is invalid!');
			ELSE
				stTimeInfos := fbAlarmManager.GetAlarmById(i).TimeInfos;
			AssertEquals(
				Expected := stTimeStruct,
				Actual := fbAlarmManager.GetAlarmById(i).TimeInfos.Acknowledged,
				Message := 'Newly registered alarm should have empty TimeInfos.Acknowledged.');
			AssertEquals(
				Expected := stTimeStruct,
				Actual := fbAlarmManager.GetAlarmById(i).TimeInfos.Activated,
				Message := 'Newly registered alarm should have empty TimeInfos.Activated.');
			AssertEquals(
				Expected := stTimeStruct,
				Actual := fbAlarmManager.GetAlarmById(i).TimeInfos.Deactivated,
				Message := 'Newly registered alarm should have empty TimeInfos.Deactivated.');
			END_IF
		END_FOR
		
		// Raise alarm
		fbAlarmManager.Actions().Raise().ById(2);
		stTimeStruct := fbAlarmManager._dateTime.CurrentTime.Value;
		stTimeStructActivation := stTimeStruct;
		alarm := fbAlarmManager.GetAlarmById(2);
		AssertEquals_WORD(
			Expected := stTimeStruct.wMilliseconds,
			Actual := alarm.TimeInfos.Activated.wMilliseconds,
			Message := 'Activation time info after raising alarm (millisecond) is incorrect.');
		AssertEquals_WORD(
			Expected := stTimeStruct.wSecond,
			Actual := alarm.TimeInfos.Activated.wSecond,
			Message := 'Activation time info after raising alarm (second) is incorrect.');
		AssertEquals_WORD(
			Expected := stTimeStruct.wMinute,
			Actual := alarm.TimeInfos.Activated.wMinute,
			Message := 'Activation time info after raising alarm (minute) is incorrect.');
		AssertEquals_WORD(
			Expected := stTimeStruct.wHour,
			Actual := alarm.TimeInfos.Activated.wHour,
			Message := 'Activation time info after raising alarm (hour) is incorrect.');
		AssertEquals_WORD(
			Expected := stTimeStruct.wDay,
			Actual := alarm.TimeInfos.Activated.wDay,
			Message := 'Activation time info after raising alarm (day) is incorrect.');
		AssertEquals_WORD(
			Expected := stTimeStruct.wMonth,
			Actual := alarm.TimeInfos.Activated.wMonth,
			Message := 'Activation time info after raising alarm (month) is incorrect.');
		AssertEquals_WORD(
			Expected := stTimeStruct.wYear,
			Actual := alarm.TimeInfos.Activated.wYear,
			Message := 'Activation time info after raising alarm (year) is incorrect.');	
		AssertEquals_WORD(
			Expected := stTimeStruct.wDayOfWeek,
			Actual := alarm.TimeInfos.Activated.wDayOfWeek,
			Message := 'Activation time info after raising alarm (day of week) is incorrect.');
			
		MEMSET(ADR(stTimeStruct),0,SIZEOF(Tc2_Utilities.TIMESTRUCT));	
		AssertEquals(
			Expected := stTimeStruct,
			Actual := fbAlarmManager.GetAlarmById(2).TimeInfos.Acknowledged,
			Message := 'When alarm is raised, the acknowledged time information should be empty.');
		AssertEquals(
			Expected := stTimeStruct,
			Actual := fbAlarmManager.GetAlarmById(2).TimeInfos.Deactivated,
			Message := 'When alarm is raised, the deactivation time information should be empty.');
		
		// Acknowledge alarm
		fbAlarmManager.Actions().Acknowledge().ById(2);
		stTimeStruct := fbAlarmManager._dateTime.CurrentTime.Value;
		stTimeStructAcnowledge := stTimeStruct;
		alarm := fbAlarmManager.GetAlarmById(2);
		
		AssertEquals_WORD(
			Expected := stTimeStruct.wMilliseconds,
			Actual := alarm.TimeInfos.Acknowledged.wMilliseconds,
			Message := 'Acknowledged time info after acknowlidging alarm (millisecond) is incorrect.');
		AssertEquals_WORD(
			Expected := stTimeStruct.wSecond,
			Actual := alarm.TimeInfos.Acknowledged.wSecond,
			Message := 'Acknowledged time info after acknowlidging alarm (second) is incorrect.');
		AssertEquals_WORD(
			Expected := stTimeStruct.wMinute,
			Actual := alarm.TimeInfos.Acknowledged.wMinute,
			Message := 'Acknowledged time info after acknowlidging alarm (minute) is incorrect.');
		AssertEquals_WORD(
			Expected := stTimeStruct.wHour,
			Actual := alarm.TimeInfos.Acknowledged.wHour,
			Message := 'Acknowledged time info after acknowlidging alarm (hour) is incorrect.');
		AssertEquals_WORD(
			Expected := stTimeStruct.wDay,
			Actual := alarm.TimeInfos.Acknowledged.wDay,
			Message := 'Acknowledged time info after acknowlidging alarm (day) is incorrect.');
		AssertEquals_WORD(
			Expected := stTimeStruct.wMonth,
			Actual := alarm.TimeInfos.Acknowledged.wMonth,
			Message := 'Acknowledged time info after acknowlidging alarm (month) is incorrect.');
		AssertEquals_WORD(
			Expected := stTimeStruct.wYear,
			Actual := alarm.TimeInfos.Acknowledged.wYear,
			Message := 'Acknowledged time info after acknowlidging alarm (year) is incorrect.');	
		AssertEquals_WORD(
			Expected := stTimeStruct.wDayOfWeek,
			Actual := alarm.TimeInfos.Acknowledged.wDayOfWeek,
			Message := 'Acknowledged time info after acknowlidging alarm (day of week) is incorrect.');
		
		MEMSET(ADR(stTimeStruct),0,SIZEOF(Tc2_Utilities.TIMESTRUCT));	
		AssertEquals(
			Expected := stTimeStruct,
			Actual := fbAlarmManager.GetAlarmById(2).TimeInfos.Deactivated,
			Message := 'When alarm is acknowledged, the deactivation time information should not change.');
		AssertEquals(
			Actual := fbAlarmManager.GetAlarmById(2).TimeInfos.Activated,
			Expected := stTimeStructActivation,
			Message := 'If alarm is acknowledged, the acivation time info should not change.');
			
		// Deactivate alarm
		fbAlarmManager.Actions().Deactivate().ById(2);
		stTimeStruct := fbAlarmManager._dateTime.CurrentTime.Value;
		alarm := fbAlarmManager.GetAlarmById(2);
		
		AssertEquals_WORD(
			Expected := stTimeStruct.wMilliseconds,
			Actual := alarm.TimeInfos.Deactivated.wMilliseconds,
			Message := 'Deactivation time info after deactivating alarm (millisecond) is incorrect.');
		AssertEquals_WORD(
			Expected := stTimeStruct.wSecond,
			Actual := alarm.TimeInfos.Deactivated.wSecond,
			Message := 'Deactivation time info after deactivating alarm (second) is incorrect.');
		AssertEquals_WORD(
			Expected := stTimeStruct.wMinute,
			Actual := alarm.TimeInfos.Deactivated.wMinute,
			Message := 'Deactivation time info after deactivating alarm (minute) is incorrect.');
		AssertEquals_WORD(
			Expected := stTimeStruct.wHour,
			Actual := alarm.TimeInfos.Deactivated.wHour,
			Message := 'Deactivation time info after deactivating alarm (hour) is incorrect.');
		AssertEquals_WORD(
			Expected := stTimeStruct.wDay,
			Actual := alarm.TimeInfos.Deactivated.wDay,
			Message := 'Deactivation time info after deactivating alarm (day) is incorrect.');
		AssertEquals_WORD(
			Expected := stTimeStruct.wMonth,
			Actual := alarm.TimeInfos.Deactivated.wMonth,
			Message := 'Deactivation time info after deactivating alarm (month) is incorrect.');
		AssertEquals_WORD(
			Expected := stTimeStruct.wYear,
			Actual := alarm.TimeInfos.Deactivated.wYear,
			Message := 'Deactivation time info after deactivating alarm (year) is incorrect.');	
		AssertEquals_WORD(
			Expected := stTimeStruct.wDayOfWeek,
			Actual := alarm.TimeInfos.Deactivated.wDayOfWeek,
			Message := 'Deactivation time info after deactivating alarm (day of week) is incorrect.');
		
		// Check that previous entries did not change	
		AssertEquals(
			Expected := stTimeStructAcnowledge,
			Actual := fbAlarmManager.GetAlarmById(2).TimeInfos.Acknowledged,
			Message := 'When alarm is acknowledged, the deactivation time information should not change.');
		AssertEquals(
			Actual := fbAlarmManager.GetAlarmById(2).TimeInfos.Activated,
			Expected := stTimeStructActivation,
			Message := 'If alarm is acknowledged, the acivation time info should not change.');
		
			
		// Activate again and confirm that acknowledge and deactivation are reset
		// Raise alarm
		fbAlarmManager.Actions().Raise().ById(2);
		MEMSET(ADR(stTimeStruct),0,SIZEOF(Tc2_Utilities.TIMESTRUCT));
		AssertEquals(
			Actual := fbAlarmManager.GetAlarmById(2).TimeInfos.Deactivated,
			Expected := stTimeStruct,
			Message := 'When alarm is re-activated, previous time information for "deactivated" should be cleared.');
		AssertEquals(
			Actual := fbAlarmManager.GetAlarmById(2).TimeInfos.Acknowledged,
			Expected := stTimeStruct,
			Message := 'When alarm is re-activated, previous time information for "acknowledged" should be cleared.');
			
		TcUnit.TEST_FINISHED();
	END_IF
END_IF
END_METHOD

METHOD Test17_RaiseUnexisitngAlarm_ExpectNoNewAlarmsActive
VAR_INPUT
END_VAR

VAR_INST
	prevAlarmActiveCount	: UINT;
	prevUnackAlarmCount		: UINT;
END_VAR
IF TcUnit.TEST_ORDERED('Test17_RaiseUnexisitngAlarm_ExpectNoNewAlarmsActive') THEN
	prevAlarmActiveCount := _alarmManager.ActiveAlarmsCount;
	prevUnackAlarmCount := _alarmManager.UnacknowledgedAlarmsCount;
	
	_alarmManager.RaiseAlarmById(24523452);
	AssertEquals_UINT(
		Actual := _alarmManager.ActiveAlarmsCount,
		Expected := prevAlarmActiveCount,
		Message := 'If an alarm that does not exist is raised, active alarms count should not change.');
		
	AssertEquals_UINT(
		Actual := _alarmManager.UnacknowledgedAlarmsCount,
		Expected := prevUnackAlarmCount,
		Message := 'If an alarm that does not exist is raised, active alarms count should not change.');
		
	_alarmManager.Actions().Raise().ById(24523452);
	AssertEquals_UINT(
		Actual := _alarmManager.ActiveAlarmsCount,
		Expected := prevAlarmActiveCount,
		Message := 'Fluent - If an alarm that does not exist is raised, active alarms count should not change.');
		
	AssertEquals_UINT(
		Actual := _alarmManager.UnacknowledgedAlarmsCount,
		Expected := prevUnackAlarmCount,
		Message := 'Fluent - If an alarm that does not exist is raised, active alarms count should not change.');
		
	TcUnit.TEST_FINISHED();
END_IF
END_METHOD

METHOD Test18_DeleteAlarm_ExpectPreviousAlarmsStillExist
VAR_INPUT
END_VAR
VAR_INST
	fbAlarmManager	: FB_AlarmManager(
		enable := TRUE, // [BOOL] - Enables alarm generation
		logger := 0, // [REFERENCE TO ZigaLibs_Core.I_LoggerEx] - optional, logger.
		timeProvider := _dateTime); //[ZigaLibs_Core.I_LocalSystemTimeProvider] - required, date time provider.
	currentAlarm	: ST_AlarmInfo;
END_VAR
IF TcUnit.TEST_ORDERED('Test18_DeleteAlarm_ExpectPreviousAlarmsStillExist') THEN
	fbAlarmManager.RegisterAlarm(1,'1','1',E_AlarmLevel.WARNING);
	fbAlarmManager.RegisterAlarm(2,'2','2',E_AlarmLevel.WARNING);
	fbAlarmManager.RegisterAlarm(3,'3','3',E_AlarmLevel.WARNING);
	fbAlarmManager.RegisterAlarm(4,'4','4',E_AlarmLevel.WARNING);
	
	fbAlarmManager.DeleteAlarm(2);
	AssertEquals_UDINT(
		Expected := 3,
		Actual := fbAlarmManager.RegisteredAlarmsCount,
		Message := 'Deleting an alarm should lower registered alarms count.');
		
	// Alarm index 1	
	currentAlarm := fbAlarmManager.GetAlarmById(1);
	AssertEquals_DINT(
		Expected := 1,
		Actual := currentAlarm.Id,
		Message := 'First alarm Id is incorrected after deleting 2nd alarm.');
	AssertEquals_STRING(
		Expected := '1',
		Actual := currentAlarm.Name,
		Message := 'First alarm Name is incorrected after deleting 2nd alarm.');
	AssertEquals_STRING(
		Expected := '1',
		Actual := currentAlarm.Message,
		Message := 'First alarm Message is incorrected after deleting 2nd alarm.');
	
	// Alarm index 2	
	// Should no longer exist
	
	AssertFalse(
		Condition := __ISVALIDREF(fbAlarmManager.GetAlarmById(2)),
		Message := 'Alarm with Id 2 should no longer exist.');
	
	
	// Alarm index 3	
	AssertTrue(
			Condition := __ISVALIDREF(fbAlarmManager.GetAlarmById(3)),
			Message := 'Alarm with Id 3 should exist.');
			
	currentAlarm := fbAlarmManager.GetAlarmById(3);
	AssertEquals_DINT(
		Expected := 3,
		Actual := currentAlarm.Id,
		Message := '3rd alarm Id is incorrected after deleting 2nd alarm.');
	AssertEquals_STRING(
		Expected := '3',
		Actual := currentAlarm.Name,
		Message := '3rd alarm Name is incorrected after deleting 2nd alarm.');
	AssertEquals_STRING(
		Expected := '3',
		Actual := currentAlarm.Message,
		Message := '3rd alarm Message is incorrected after deleting 2nd alarm.');
		
	// Alarm index 4		
	currentAlarm := fbAlarmManager.GetAlarmById(4);
	AssertEquals_DINT(
		Expected := 4,
		Actual := currentAlarm.Id,
		Message := '4th alarm Id is incorrected after deleting 2nd alarm.');
	AssertEquals_STRING(
		Expected := '4',
		Actual := currentAlarm.Name,
		Message := '4th alarm Name is incorrected after deleting 2nd alarm.');
	AssertEquals_STRING(
		Expected := '4',
		Actual := currentAlarm.Message,
		Message := '4th alarm Message is incorrected after deleting 2nd alarm.');
		
	TcUnit.TEST_FINISHED();
END_IF
END_METHOD

METHOD Test19_DeleteUnexistingAlarm_ExpectNoChangesToExistingAlarms
VAR_INPUT
END_VAR
VAR_INST
	fbAlarmManager	: FB_AlarmManager(
		enable := TRUE, // [BOOL] - Enables alarm generation
		logger := 0, // [REFERENCE TO ZigaLibs_Core.I_LoggerEx] - optional, logger.
		timeProvider := _dateTime); //[ZigaLibs_Core.I_LocalSystemTimeProvider] - required, date time provider.
	currentAlarm	: ST_AlarmInfo;
	emptyAlarm		: ST_AlarmInfo;
END_VAR
IF TcUnit.TEST_ORDERED('Test19_DeleteUnexistingAlarm_ExpectNoChangesToExistingAlarms') THEN
	fbAlarmManager.RegisterAlarm(1,'1','1',E_AlarmLevel.ERROR);
	fbAlarmManager.RegisterAlarm(2,'2','2',E_AlarmLevel.INFO);
	fbAlarmManager.RegisterAlarm(3,'3','3',E_AlarmLevel.WARNING);
	fbAlarmManager.RegisterAlarm(4,'4','4',E_AlarmLevel.WARNING);
	
	// Delete unexisting alarm, expect no changes.
	fbAlarmManager.DeleteAlarm(0);
	AssertEquals_UDINT(
		Expected := 4,
		Actual := fbAlarmManager.RegisteredAlarmsCount,
		Message := 'Deleting unexisting alarm should not change registered alarms count.');
		
	currentAlarm := fbAlarmManager.GetAlarmById(1);
	AssertEquals_DINT(
		Expected := 1,
		Actual := currentAlarm.Id,
		Message := 'First alarm Id is incorrected after deleting unexisting alarm.');
	AssertEquals_STRING(
		Expected := '1',
		Actual := currentAlarm.Name,
		Message := 'First alarm Name is incorrected after deleting unexisting alarm.');
	AssertEquals_STRING(
		Expected := '1',
		Actual := currentAlarm.Message,
		Message := 'First alarm Message is incorrected after deleting unexisting alarm.');
		
	currentAlarm := fbAlarmManager.GetAlarmById(2);
	AssertEquals_DINT(
		Expected := 2,
		Actual := currentAlarm.Id,
		Message := '2nd alarm Id is incorrected after deleting unexisting alarm.');
	AssertEquals_STRING(
		Expected := '2',
		Actual := currentAlarm.Name,
		Message := '2nd alarm Name is incorrected after deleting unexisting alarm.');
	AssertEquals_STRING(
		Expected := '2',
		Actual := currentAlarm.Message,
		Message := '2nd alarm Message is incorrected after deleting unexisting alarm.');
		
	currentAlarm := fbAlarmManager.GetAlarmById(3);
	AssertEquals_DINT(
		Expected := 3,
		Actual := currentAlarm.Id,
		Message := '3rd alarm Id is incorrected after deleting unexisting alarm.');
	AssertEquals_STRING(
		Expected := '3',
		Actual := currentAlarm.Name,
		Message := '3rd alarm Name is incorrected after deleting unexisting alarm.');
	AssertEquals_STRING(
		Expected := '3',
		Actual := currentAlarm.Message,
		Message := '3rd alarm Message is incorrected after deleting unexisting alarm.');
		
	currentAlarm := fbAlarmManager.GetAlarmById(4);
	AssertEquals_DINT(
		Expected := 4,
		Actual := currentAlarm.Id,
		Message := '4th alarm Id is incorrected after deleting unexisting alarm.');
	AssertEquals_STRING(
		Expected := '4',
		Actual := currentAlarm.Name,
		Message := '4th alarm Name is incorrected after deleting unexisting alarm.');
	AssertEquals_STRING(
		Expected := '4',
		Actual := currentAlarm.Message,
		Message := '4th alarm Message is incorrected after deleting unexisting alarm.');
		
	TcUnit.TEST_FINISHED();
END_IF
END_METHOD

METHOD Test20_DeleteAll
VAR_INST
	fbAlarmManager	: FB_AlarmManager(
		enable := TRUE,
		logger := 0,
		timeProvider := _dateTime);
	currentAlarm
	: ST_AlarmInfo;
	emptyAlarm		: ST_AlarmInfo;
	i	: INT;
END_VAR
TcUnit.TEST('Test20_DeleteAll');

FOR i := 0 TO 5 BY 1 DO
	fbAlarmManager.RegisterAlarm(i, TO_STRING(i), TO_STRING(i), E_AlarmLevel.ERROR);
	fbAlarmManager.Actions().Raise().ById(i);
END_FOR

fbAlarmManager.DeleteAll();
AssertEquals_DINT(0, fbAlarmManager.RegisteredAlarmsCount, 'Deleteing all alarms should result in the registered alarm count being 0.');
AssertEquals_DINT(0, fbAlarmMAnager.ActiveAlarmsCount, 'Deleting all alarms should result in active alarms count being 0');
AssertEquals_DINT(0, fbAlarmManager.UnacknowledgedAlarmsCount, 'Deleting all alarms should result in unacknowledged alarms count being 0');
AssertFalse(__ISVALIDREF(fbAlarmManager.GetAlarmById(1)), 'Attempting to retrive an alarm when they have all been deleted should return an empty reference.');

TcUnit.TEST_FINISHED();
END_METHOD

END_FUNCTION_BLOCK

// TESTS/PRG_TESTS
PROGRAM INTERNAL PRG_TESTS

(* Instantiate test suites here. Naming convention for tests should be a suffix with _Tests.
Good practice for creating test methods is to end them with _test as well. *)
VAR
	AlarmManagerTests	: FB_AlarmManager_Tests;
END_VAR

// Run tests in parallel
//TcUnit.RUN();

// Run tests in sequence, one after the other.
TcUnit.RUN_IN_SEQUENCE();

END_PROGRAM
